{attribute 'qualified_only'}
{attribute 'strict'}
{attribute 'to_string'}
TYPE ST_EMoverLoadType :
(
	Wellplate := 1,
	PipetteTips:=2,
	Gripper:=3
);
END_TYPE

(* stored: Version 1.1.0.1
   DUT ST_EMoverLoadType: Id {b001b95b-474a-4457-938f-12956e7181f7} *)
